// TIA Portal V20 export
VAR_GLOBAL   // PLC tag table "Default tag table"
   Tag_3 AT %IB0 : Byte;
   System_Byte AT %MB1 : Byte;   //    {ExternalAccessible false, ExternalVisible false, ExternalWritable false}
   FirstScan AT %M1.0 : Bool;   //    {ExternalAccessible false, ExternalVisible false, ExternalWritable false}
   DiagStatusUpdate AT %M1.1 : Bool;   //    {ExternalAccessible false, ExternalVisible false, ExternalWritable false}
   AlwaysTRUE AT %M1.2 : Bool;   //    {ExternalAccessible false, ExternalVisible false, ExternalWritable false}
   AlwaysFALSE AT %M1.3 : Bool;   //    {ExternalAccessible false, ExternalVisible false, ExternalWritable false}
   Clock_Byte AT %MB0 : Byte;   //    {ExternalAccessible false, ExternalVisible false, ExternalWritable false}
   Clock_10Hz AT %M0.0 : Bool;   //    {ExternalAccessible false, ExternalVisible false, ExternalWritable false}
   Clock_5Hz AT %M0.1 : Bool;   //    {ExternalAccessible false, ExternalVisible false, ExternalWritable false}
   "Clock_2.5Hz" AT %M0.2 : Bool;   //    {ExternalAccessible false, ExternalVisible false, ExternalWritable false}
   Clock_2Hz AT %M0.3 : Bool;   //    {ExternalAccessible false, ExternalVisible false, ExternalWritable false}
   "Clock_1.25Hz" AT %M0.4 : Bool;   //    {ExternalAccessible false, ExternalVisible false, ExternalWritable false}
   Clock_1Hz AT %M0.5 : Bool;   //    {ExternalAccessible false, ExternalVisible false, ExternalWritable false}
   "Clock_0.625Hz" AT %M0.6 : Bool;   //    {ExternalAccessible false, ExternalVisible false, ExternalWritable false}
   "Clock_0.5Hz" AT %M0.7 : Bool;   //    {ExternalAccessible false, ExternalVisible false, ExternalWritable false}
   Init AT %M100.0 : Bool;   //    {ExternalAccessible false, ExternalVisible false, ExternalWritable false}
   Tag_1 AT %M500.0 : Bool;   //    {ExternalAccessible false, ExternalVisible false, ExternalWritable false}
   InitByte AT %MB300 : Byte;   //    {ExternalAccessible false, ExternalVisible false, ExternalWritable false}
   Tag_2 AT %M500.1 : Bool;   //    {ExternalAccessible false, ExternalVisible false, ExternalWritable false}
   Load AT %M800.0 : Bool;
   Tag_4 AT %M8000.0 : Bool;
   Reset AT %M8000.1 : Bool;
   Test_MCS AT %MD8004 : Real;
   Test_ACS AT %MD8008 : Real;
   Tag_6 AT %M9000.0 : Bool;
   ParaDB2CSV AT %M8000.2 : Bool;
   Tag_5 AT %M8000.3 : Bool;
   CompleteMm AT %M8000.4 : Bool;
   Tag_7 AT %M300.0 : Bool;
   Tag_8 AT %M301.0 : Bool;
   Tag_9 AT %M301.1 : Bool;
   Tic AT %M302.0 : Bool;
   PPipOffDlyMm AT %MD308 : Real;
   Tac AT %M302.1 : Bool;
   Tag_10 AT %MD500 : Real;
   Tag_11 AT %MD504 : Real;
   Tag_12 AT %MD508 : Real;
   Tag_13 AT %MD512 : Real;
   Tag_14 AT %M600.1 : Bool;
   TorqueCal AT %MD600 : Real;
   FLD_Normal_PCR AT %I1205.5 : Bool;
   FLD_Normal_TBR AT %I1213.5 : Bool;
   FLD_Normal_PCR_Intensity AT %I1205.7 : Bool;
   FLD_Normal_TBR_Intensity AT %I1213.7 : Bool;
   "i1202.2" AT %I1202.2 : Bool;
   "i1202.3" AT %I1202.3 : Bool;
   "i1202.4" AT %I1202.4 : Bool;
   "i1202.5" AT %I1202.5 : Bool;
   "i1202.6" AT %I1202.6 : Bool;
END_VAR
VAR_GLOBAL CONSTANT   // user constants
   SensorCheck_FallingEdge : USInt := 0;
   SensorCheck_Off : USInt := 3;
   SensorCheck_On : USInt := 2;
   SensorCheck_RisingEdge : USInt := 1;
   IDLE : UInt := 0;
   JOG_POS : UInt := 100;
   JOG_SPD : UInt := 101;
   SPD_CTRL : UInt := 200;
   HOMING : UInt := 300;
   HOMEING_OFFSET : UInt := 301;
   ABS_POS : UInt := 400;
   REL_POS : UInt := 401;
   BRK_OPEN : UInt := 700;
END_VAR
